(* CODESYS project GVL_AXIS.gvl.xml

Project tree, tasks and I/O mapping:
  global variables GVL_AXIS
*)

// GVL_AXIS
{attribute 'qualified_only'}
VAR_GLOBAL
	arrAxis: ARRAY [1..3] OF ST_AXIS; 
END_VAR
